// TIA Portal V17 export
// export: Created 2024-08-11T17:53:04.8340159Z, ExportSetting WithDefaults, DisplayName Totally Integrated Automation Portal, DisplayVersion V17 Update 5, DisplayName TIA Portal Openness, DisplayVersion V17 Update 5, DisplayName TIA Portal Version Control Interface, DisplayVersion V17, DisplayName SINAMICS Startdrive Advanced, DisplayVersion V17 SP1, DisplayName SINAMICS Startdrive G130, G150, S120, S150, SINAMICS MV, S210, DisplayVersion V17 SP1, DisplayName SINAMICS Startdrive G110M, G120, G120C, G120D, G120P, G115D, DisplayVersion V17 SP1, DisplayName STEP 7 Professional, DisplayVersion V17 Update 5, DisplayName STEP 7 Safety, DisplayVersion V17, DisplayName WinCC Advanced / Unified PC, DisplayVersion V17 Update 5
ORGANIZATION_BLOCK "Main"   // OB1, LAD, ProgramCycle
TITLE = "Main Program Sweep (Cycle)"
{ S7_Optimized_Access := 'TRUE' }
VERSION : 0.1
// stored: AutoNumber true, IsIECCheckEnabled false, SetENOAutomatically false
   VAR_INPUT
      Initial_Call : Bool;   // Initial call of this OB
      Remanence : Bool;   // =True, if remanent data are available
   END_VAR
BEGIN

REGION Network 1: ----------[MODBUS COMMUNICATION SETTING UP]----------
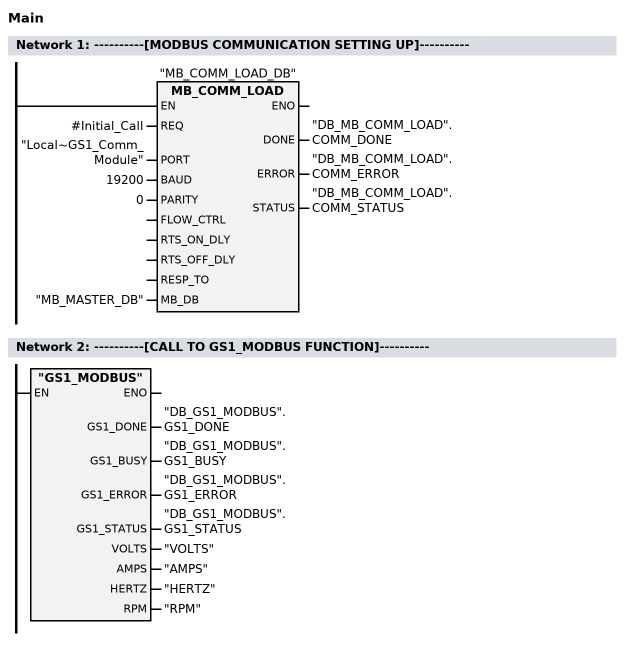
   RUNG wire#powerrail
      "MB_COMM_LOAD_DB".MB_COMM_LOAD(REQ := #Initial_Call, PORT := "Local~GS1_Comm_Module", BAUD := 19200, PARITY := 0, FLOW_CTRL :=, RTS_ON_DLY :=, RTS_OFF_DLY :=, RESP_TO :=, MB_DB := "MB_MASTER_DB", DONE => "DB_MB_COMM_LOAD".COMM_DONE, ERROR => "DB_MB_COMM_LOAD".COMM_ERROR, STATUS => "DB_MB_COMM_LOAD".COMM_STATUS)
   END_RUNG
   // the same network as SCL:
   "MB_COMM_LOAD_DB"(REQ := #Initial_Call,   // MB_COMM_LOAD
                     PORT := "Local~GS1_Comm_Module",
                     BAUD := 19200,
                     PARITY := 0,
                     MB_DB := "MB_MASTER_DB",
                     DONE => "DB_MB_COMM_LOAD".COMM_DONE,
                     ERROR => "DB_MB_COMM_LOAD".COMM_ERROR,
                     STATUS => "DB_MB_COMM_LOAD".COMM_STATUS);
END_REGION

REGION Network 2: ----------[CALL TO GS1_MODBUS FUNCTION]----------
   RUNG wire#powerrail
      "GS1_MODBUS"(GS1_DONE => "DB_GS1_MODBUS".GS1_DONE, GS1_BUSY => "DB_GS1_MODBUS".GS1_BUSY, GS1_ERROR => "DB_GS1_MODBUS".GS1_ERROR, GS1_STATUS => "DB_GS1_MODBUS".GS1_STATUS, VOLTS => "VOLTS", AMPS => "AMPS", HERTZ => "HERTZ", RPM => "RPM")
   END_RUNG
   // the same network as SCL:
   "GS1_MODBUS"(GS1_DONE => "DB_GS1_MODBUS".GS1_DONE,
                GS1_BUSY => "DB_GS1_MODBUS".GS1_BUSY,
                GS1_ERROR => "DB_GS1_MODBUS".GS1_ERROR,
                GS1_STATUS => "DB_GS1_MODBUS".GS1_STATUS,
                VOLTS => "VOLTS",
                AMPS => "AMPS",
                HERTZ => "HERTZ",
                RPM => "RPM");
END_REGION
END_ORGANIZATION_BLOCK
